{region "Read"}
5:
{region "Start Qiescent Mode"}
	fb103StartQuiescentMode(bStart := TRUE,
							eAddressType := Tc3_DALI.E_DALIAddressType.Broadcast,
							eCommandPriority := Tc3_DALI.E_DALICommandPriority.Middle);
	IF (NOT fb103StartQuiescentMode.bBusy) THEN
		fb103StartQuiescentMode(bStart := FALSE);
		nStep := 10;
	END_IF
{endregion}
10:
{region "Query Instance Error"}
	fb103QueryInstanceError(bStart := TRUE,
							nAddress := nAddress,
							eAddressType := Tc3_DALI.E_DALIAddressType.Short,
							nInstanceAddress := nInstanceAddress,
							eInstanceAddressType := Tc3_DALI.E_DALIInstanceAddressType.InstanceNumber,
							eCommandPriority := Tc3_DALI.E_DALICommandPriority.Middle,
							nInstanceError => nInstanceError);
	IF (NOT fb103QueryInstanceError.bBusy) THEN
		fb103QueryInstanceError(bStart := FALSE);
		nStep := 20;
	END_IF
{endregion}
20:
{region "Query Instance Status"}
	fb103QueryInstanceStatus(	bStart := TRUE,
								nAddress := nAddress,
								eAddressType := Tc3_DALI.E_DALIAddressType.Short,
								nInstanceAddress := nInstanceAddress,
								eInstanceAddressType := Tc3_DALI.E_DALIInstanceAddressType.InstanceNumber,
								eCommandPriority := Tc3_DALI.E_DALICommandPriority.Middle);
	IF (NOT fb103QueryInstanceStatus.bBusy) THEN
		fb103QueryInstanceStatus(bStart := FALSE);
		IF (fb103QueryInstanceStatus.nInstanceStatus.1) THEN
			bEnable := TRUE;
		END_IF
			nStep := 30;
	END_IF
30:
{region "Query Resolution"}
	fb103QueryResolution(	bStart := TRUE,
							nAddress := nAddress,
							eAddressType := Tc3_DALI.E_DALIAddressType.Short,
							nInstanceAddress := nInstanceAddress,
							eInstanceAddressType := Tc3_DALI.E_DALIInstanceAddressType.InstanceNumber,
							eCommandPriority := Tc3_DALI.E_DALICommandPriority.Middle,
							nResolution => nResolution);
	IF (NOT fb103QueryResolution.bBusy) THEN
		fb103QueryResolution(bStart := FALSE);
		nStep := 40;
	END_IF
{endregion}
40:
{region "Query Input Value"}
	fb103QueryInputValue(	bStart := TRUE,
							nAddress := nAddress,
							eAddressType:= Tc3_DALI.E_DALIAddressType.Short,
							nInstanceAddress := nInstanceAddress,
							eInstanceAddressType := Tc3_DALI.E_DALIInstanceAddressType.InstanceNumber,
							eCommandPriority := Tc3_DALI.E_DALICommandPriority.Middle,
							nResolution := nResolution,
							nInputValue => nInputValue);
	IF (NOT fb103QueryInputValue.bBusy) THEN
		fb103QueryInputValue(bStart := FALSE);
		nStep := 50;
	END_IF
{endregion}
50:
{region "Query Event Scheme"}
	fb103QueryEventScheme(	bStart := TRUE,
							nAddress := nAddress,
							eAddressType := Tc3_DALI.E_DALIAddressType.Short,
							nInstanceAddress := nInstanceAddress,
							eInstanceAddressType := Tc3_DALI.E_DALIInstanceAddressType.InstanceNumber,
							eCommandPriority := Tc3_DALI.E_DALICommandPriority.Middle,
							eEventScheme => eEventScheme);
	IF (NOT fb103QueryEventScheme.bBusy) THEN
		fb103QueryEventScheme(bStart := FALSE);
		nStep := 60;
	END_IF
{endregion}
60:
{region "Query Event Filter"}
	fb103QueryEventFilter(	bStart := TRUE,
							nAddress := nAddress,
							eAddressType := Tc3_DALI.E_DALIAddressType.Short,
							nInstanceAddress := nInstanceAddress,
							eInstanceAddressType := Tc3_DALI.E_DALIInstanceAddressType.InstanceNumber,
							eCommandPriority := Tc3_DALI.E_DALICommandPriority.Middle,
							nEventFilter => nEventFilter);
	IF (NOT fb103QueryEventFilter.bBusy) THEN
		fb103QueryEventFilter(bStart := FALSE);
		bPositionEventEnabled := nEventFilter.0;
		nStep := 70;
	END_IF
{endregion}
70:
{region "Query Report Timer"}
	fb302QueryReportTimer(	bStart := TRUE,
							nAddress := nAddress,
							eAddressType := Tc3_DALI.E_DALIAddressType.Short,
							nInstanceAddress := nInstanceAddress,
							eInstanceAddressType := Tc3_DALI.E_DALIInstanceAddressType.InstanceNumber,
							eCommandPriority := Tc3_DALI.E_DALICommandPriority.Middle,
							nReport => nReport);
	IF (NOT fb302QueryReportTimer.bBusy) THEN
		fb302QueryReportTimer(bStart := FALSE);
		nStep := 80;
	END_IF
{endregion}
80:
{region "Query Deadtime Timer"}
	fb302QueryDeadtimeTimer(bStart := TRUE,
							nAddress := nAddress,
							eAddressType := Tc3_DALI.E_DALIAddressType.Short,
							nInstanceAddress := nInstanceAddress,
							eInstanceAddressType := Tc3_DALI.E_DALIInstanceAddressType.InstanceNumber,
							eCommandPriority := Tc3_DALI.E_DALICommandPriority.Middle);
	nDeadtime := (fb302QueryDeadtimeTimer.nDeadtime * 50);
	IF (NOT fb302QueryDeadtimeTimer.bBusy) THEN
		fb302QueryDeadtimeTimer(bStart := FALSE);
		nStep := 90;
	END_IF
{endregion}
90:
	{region "Query Deadtime Timer"}
	fb302QuerySwitch(	bStart := TRUE,
						nAddress := nAddress,
						eAddressType := Tc3_DALI.E_DALIAddressType.Short,
						nInstanceAddress := nInstanceAddress,
						eInstanceAddressType := Tc3_DALI.E_DALIInstanceAddressType.InstanceNumber,
						eCommandPriority := Tc3_DALI.E_DALICommandPriority.Middle,
						bSwitch => bSwitch);
	IF (NOT fb302QueryDeadtimeTimer.bBusy) THEN
		fb302QueryDeadtimeTimer(bStart := FALSE);
		nStep := 100;
	END_IF
{endregion}
100:
{region "Query Event Priority"}
	fb103QueryEventPriority(bStart := TRUE,
							nAddress := nAddress,
							eAddressType := Tc3_DALI.E_DALIAddressType.Short,
							nInstanceAddress := nInstanceAddress,
							eInstanceAddressType := Tc3_DALI.E_DALIInstanceAddressType.InstanceNumber,
							eCommandPriority := Tc3_DALI.E_DALICommandPriority.Middle,
							eEventPriority => eEventPriority);
	IF (NOT fb103QueryEventPriority.bBusy) THEN
		fb103QueryEventPriority(bStart := FALSE);
		nStep := 110;
	END_IF 
{endregion}
110:
{region "Stop Qiescent Mode"}
	fb103StopQuiescentMode(	bStart := TRUE,
							eAddressType := Tc3_DALI.E_DALIAddressType.Broadcast,
							eCommandPriority := Tc3_DALI.E_DALICommandPriority.Middle);
	IF (NOT fb103StopQuiescentMode.bBusy) THEN
		fb103StopQuiescentMode(bStart := FALSE);
		nStep := 0;
	END_IF
{endregion}
{region "Write"}
1000:
{region "Enable or Disable Instance"}
	IF (bEnable) THEN
		fb103EnableInstance(bStart := TRUE,
							nAddress := nAddress,
							eAddressType := Tc3_DALI.E_DALIAddressType.Short,
							nInstanceAddress := nInstanceAddress,
							eInstanceAddressType := Tc3_DALI.E_DALIInstanceAddressType.InstanceNumber,
							eCommandPriority := Tc3_DALI.E_DALICommandPriority.Middle);
		IF (NOT fb103EnableInstance.bBusy) THEN
			fb103EnableInstance(bStart := FALSE);
			nStep := 1010;
		END_IF
	ELSE
		fb103DisableInstance(	bStart := TRUE,
								nAddress := nAddress,
								eAddressType := Tc3_DALI.E_DALIAddressType.Short,
								nInstanceAddress := nInstanceAddress,
								eInstanceAddressType := Tc3_DALI.E_DALIInstanceAddressType.InstanceNumber,
								eCommandPriority := Tc3_DALI.E_DALICommandPriority.Middle);
		IF (NOT fb103DisableInstance.bBusy) THEN
			fb103DisableInstance(bStart := FALSE);
			nStep := 0;
		END_IF
	END_IF
{endregion}
1010:
{region "Set Event Scheme"}
	fb103SetEventScheme(bStart := TRUE,
						nAddress := nAddress,
						eAddressType := Tc3_DALI.E_DALIAddressType.Short,
						nInstanceAddress := nInstanceAddress,
						eInstanceAddressType := Tc3_DALI.E_DALIInstanceAddressType.InstanceNumber,
						eCommandPriority := Tc3_DALI.E_DALICommandPriority.Middle,
						eEventScheme := eEventScheme);
	IF (NOT fb103SetEventScheme.bBusy) THEN
		fb103SetEventScheme(bStart := FALSE);
		nStep := 1020;
	END_IF
{endregion}
1020:
{region "Set Event Filter"}
	nEventFilter.0 := bPositionEventEnabled;
	fb103SetEventFilter(bStart := TRUE,
						nAddress := nAddress,
						eAddressType := Tc3_DALI.E_DALIAddressType.Short,
						nInstanceAddress := nInstanceAddress,
						eInstanceAddressType := Tc3_DALI.E_DALIInstanceAddressType.InstanceNumber,
						eCommandPriority := Tc3_DALI.E_DALICommandPriority.Middle,
						nEventFilter := nEventFilter);
	IF (NOT fb103SetEventFilter.bBusy) THEN
		fb103SetEventFilter(bStart := FALSE);
		nStep := 1030;
	END_IF
{endregion}
1030:
{region "Set Report Timer"}
	IF (bNoReportTimer) THEN
		nStep := 1040;
	ELSE
		fb302SetReportTimer(bStart := TRUE,
							nAddress := nAddress,
							eAddressType := Tc3_DALI.E_DALIAddressType.Short,
							nInstanceAddress := nInstanceAddress,
							eInstanceAddressType := Tc3_DALI.E_DALIInstanceAddressType.InstanceNumber,
							eCommandPriority := Tc3_DALI.E_DALICommandPriority.Middle,
							nReport := nReport);
		IF (NOT fb302SetReportTimer.bBusy) THEN
			fb302SetReportTimer(bStart := FALSE);
			nStep := 1040;
		END_IF
	END_IF
{endregion}
1040:
{region "Set Deadtime Timer"}
	IF (bNoDeadtimeTimer) THEN
		nStep := 1050;
	ELSE
		fb302SetDeadtimeTimer(	bStart := TRUE,
								nAddress := nAddress,
								eAddressType := Tc3_DALI.E_DALIAddressType.Short,
								nInstanceAddress := nInstanceAddress,
								eInstanceAddressType := Tc3_DALI.E_DALIInstanceAddressType.InstanceNumber,
								eCommandPriority := Tc3_DALI.E_DALICommandPriority.Middle,
								nDeadtime := TO_BYTE(nDeadtime / 50));
		IF (NOT fb302SetDeadtimeTimer.bBusy) THEN
			fb302SetDeadtimeTimer(bStart := FALSE);
			nStep := 1050;
		END_IF
	END_IF
{endregion}
1050:
{region "Set Event Priority"}
	fb103SetEventPriority(	bStart := TRUE,
							nAddress := nAddress,
							eAddressType := Tc3_DALI.E_DALIAddressType.Short,
							nInstanceAddress := nInstanceAddress,
							eInstanceAddressType := Tc3_DALI.E_DALIInstanceAddressType.InstanceNumber,
							eCommandPriority := Tc3_DALI.E_DALICommandPriority.Middle,
							eEventPriority := eEventPriority);
	IF (NOT fb103SetEventPriority.bBusy) THEN
		fb103SetEventPriority(bStart := FALSE);
		nStep := 0;
	END_IF
{endregion}
END_CASE
{endregion}

END_FUNCTION_BLOCK

// ---- POUs/DALI/DALI_Setup/FBs/FB_Part303OccupancySensor.TcPOU
FUNCTION_BLOCK FB_Part303OccupancySensor
VAR_INPUT
	ipDALICommunication			:	I_DALICommunication;
END_VAR
VAR_OUTPUT
	bBusy						:	BOOL;
END_VAR
VAR
{region "Visu"}
	sInputValue					:	STRING (50);
	nInstanceError				:	BYTE;
	nResolution					:	BYTE;
	eEventScheme				:	E_DALIEventScheme;
	nEventFilter				:	DWORD;
	nHold						:	UINT(1..2538);
	nHoldIntern					:	BYTE;
	nReport						:	BYTE(0..255);
	nDeadtime					:	UINT(0..12750);
	nDeadtimeIntern				:	BYTE;
	sCatching					:	STRING (20);
	bEnable						:	BOOL;
	bCancelHoldTimer			:	BOOL;
	bCatchmovement				:	BOOL;
	bRead						:	BOOL;
	bWrite						:	BOOL;
	bOccupied					:	BOOL;
	bVacant						:	BOOL;
	bRepeat						:	BOOL;
	bMovement					:	BOOL;
	bNoMovement					:	BOOL;
	bNoHoldTimer				:	BOOL;
	bNoReportTimer				:	BOOL;
	bNoDeadtimeTimer			:	BOOL;
	eEventPriority				:	E_DALIEventPriority := E_DALIEventPriority.MiddleLow;
{endregion}
	nStep						:	INT;
	nAddress					:	BYTE;
	nInstanceAddress			:	BYTE;
	bHideWaitSymbol				:	BOOL := TRUE;

	fb103StartQuiescentMode		:	FB_DALI103StartQuiescentMode(0);
	fb103StopQuiescentMode		:	FB_DALI103StopQuiescentMode(0);
	fb103QueryInstanceError		:	FB_DALI103QueryInstanceError(0);
	fb103QueryInstanceStatus	:	FB_DALI103QueryInstanceStatus(0);
	fb103QueryResolution		:	FB_DALI103QueryResolution(0);
	fb103QueryInputValue 		:	FB_DALI103QueryInputValue(0);
	fb103QueryEventScheme 		:	FB_DALI103QueryEventScheme(0);
	fb103QueryEventFilter 		:	FB_DALI103QueryEventFilter(0);
	fb103QueryEventPriority		:	FB_DALI103QueryEventPriority(0);
	fb303QueryCatching			:	FB_DALI303QueryCatching(0);
	fb303QueryHoldTimer			:	FB_DALI303QueryHoldTimer(0);
	fb303QueryReportTimer		:	FB_DALI303QueryReportTimer(0);
	fb303QueryDeadtimeTimer		:	FB_DALI303QueryDeadtimeTimer(0);
	fb103EnableInstance			:	FB_DALI103EnableInstance(0);
	fb103DisableInstance		:	FB_DALI103DisableInstance(0);
	fb103SetEventScheme			:	FB_DALI103SetEventScheme(0);
	fb103SetEventFilter			:	FB_DALI103SetEventFilter(0);
	fb103SetEventPriority		:	FB_DALI103SetEventPriority(0);
	fb303SetHoldTimer			:	FB_DALI303SetHoldTimer(0);
	fb303SetReportTimer			:	FB_DALI303SetReportTimer(0);
	fb303SetDeadtimeTimer		:	FB_DALI303SetDeadtimeTimer(0);
	fb303CancelHoldTimer		:	FB_DALI303CancelHoldTimer(0);
	fb303CatchMovement			:	FB_DALI303CatchMovement(0);
END_VAR

{region "Detect Commands"}
IF (bRead AND (nStep = 0)) THEN
	nStep := 5;
	bRead := FALSE;
	bHideWaitSymbol := FALSE;
END_IF

IF (bWrite AND (nStep = 0)) THEN
	nStep := 1000;
	bWrite := FALSE;
	bHideWaitSymbol := FALSE;
END_IF
{endregion}
{region "Manage Dialog Selection}
IF (nStep = 0) THEN
	bBusy := FALSE;
ELSE
	bBusy := TRUE;
END_IF
{endregion}
{region "Execute Commands"}
CASE nStep OF
0:
{region "Init"}
	bRead := FALSE;
	bWrite := FALSE;
	bHideWaitSymbol := TRUE;

	fb103StartQuiescentMode.ipDALICommunication := ipDALICommunication;
	fb103StopQuiescentMode.ipDALICommunication := ipDALICommunication;
	fb103QueryInstanceError.ipDALICommunication := ipDALICommunication;
	fb103QueryInstanceStatus.ipDALICommunication := ipDALICommunication;
	fb103QueryResolution.ipDALICommunication := ipDALICommunication;
	fb103QueryInputValue.ipDALICommunication := ipDALICommunication;
	fb103QueryEventScheme.ipDALICommunication := ipDALICommunication;
	fb103QueryEventFilter.ipDALICommunication := ipDALICommunication;
	fb103QueryEventPriority.ipDALICommunication := ipDALICommunication;
	fb303QueryCatching.ipDALICommunication := ipDALICommunication;
	fb303QueryHoldTimer.ipDALICommunication := ipDALICommunication;
	fb303QueryReportTimer.ipDALICommunication := ipDALICommunication;
	fb303QueryDeadtimeTimer.ipDALICommunication := ipDALICommunication;
	fb103EnableInstance.ipDALICommunication := ipDALICommunication;
	fb103DisableInstance.ipDALICommunication := ipDALICommunication;
	fb103SetEventScheme.ipDALICommunication := ipDALICommunication;
	fb103SetEventFilter.ipDALICommunication := ipDALICommunication;
	fb103SetEventPriority.ipDALICommunication := ipDALICommunication;
	fb303SetHoldTimer.ipDALICommunication := ipDALICommunication;
	fb303SetReportTimer.ipDALICommunication := ipDALICommunication;
	fb303SetDeadtimeTimer.ipDALICommunication := ipDALICommunication;
	fb303CancelHoldTimer.ipDALICommunication := ipDALICommunication;
	fb303CatchMovement.ipDALICommunication := ipDALICommunication;
{endregion}
{region "Read"}
5:
{region "Start Qiescent Mode"}
	fb103StartQuiescentMode(bStart := TRUE,
							eAddressType := Tc3_DALI.E_DALIAddressType.Broadcast,
							eCommandPriority := Tc3_DALI.E_DALICommandPriority.Middle);
	IF (NOT fb103StartQuiescentMode.bBusy) THEN
		fb103StartQuiescentMode(bStart:= FALSE);
		nStep := 10;
	END_IF
{endregion}
10:
{region "Query Instance Error"}
	fb103QueryInstanceError(bStart := TRUE,
							nAddress := nAddress,
							eAddressType := Tc3_DALI.E_DALIAddressType.Short,
							nInstanceAddress := nInstanceAddress,
							eInstanceAddressType := Tc3_DALI.E_DALIInstanceAddressType.InstanceNumber,
							eCommandPriority := Tc3_DALI.E_DALICommandPriority.Middle,
							nInstanceError => nInstanceError);
	IF (NOT fb103QueryInstanceError.bBusy) THEN
		fb103QueryInstanceError(bStart := FALSE);
		nStep := 20;
	END_IF
{endregion}
20:
{region "Query Instance Status"}
	fb103QueryInstanceStatus(	bStart := TRUE,
								nAddress := nAddress,
								eAddressType := Tc3_DALI.E_DALIAddressType.Short,
								nInstanceAddress := nInstanceAddress,
								eInstanceAddressType := Tc3_DALI.E_DALIInstanceAddressType.InstanceNumber,
								eCommandPriority := Tc3_DALI.E_DALICommandPriority.Middle);
	IF (NOT fb103QueryInstanceStatus.bBusy) THEN
		fb103QueryInstanceStatus(bStart := FALSE);
		IF (fb103QueryInstanceStatus.nInstanceStatus.1) THEN
			bEnable := TRUE;
		END_IF
		nStep := 30;
	END_IF
30:
{region "Query Resolution"}
	fb103QueryResolution(	bStart := TRUE,
							nAddress := nAddress,
							eAddressType := Tc3_DALI.E_DALIAddressType.Short,
							nInstanceAddress := nInstanceAddress,
							eInstanceAddressType := Tc3_DALI.E_DALIInstanceAddressType.InstanceNumber,
							eCommandPriority := Tc3_DALI.E_DALICommandPriority.Middle,
							nResolution => nResolution);
	IF (NOT fb103QueryResolution.bBusy) THEN
		fb103QueryResolution(bStart := FALSE);
		nStep := 40;
	END_IF
{endregion}
40:
{region "Query Input Value"}
	fb103QueryInputValue(	bStart := TRUE,
							nAddress := nAddress,
							eAddressType := Tc3_DALI.E_DALIAddressType.Short,
							nInstanceAddress := nInstanceAddress,
							eInstanceAddressType := Tc3_DALI.E_DALIInstanceAddressType.InstanceNumber,
							eCommandPriority := Tc3_DALI.E_DALICommandPriority.Middle,
							nResolution := nResolution);
	IF (NOT fb103QueryInputValue.bBusy) THEN
		fb103QueryInputValue(bStart:= FALSE);
		IF (fb103QueryInputValue.nInputValue = 0) THEN
			sInputValue := 'Vacant and no movement';
		ELSIF (fb103QueryInputValue.nInputValue = 1) THEN
			sInputValue := 'Vacant and movement';
		ELSIF (fb103QueryInputValue.nInputValue = 2) THEN
			sInputValue := 'Occupied and no movement';
		ELSIF (fb103QueryInputValue.nInputValue = 3) THEN
			sInputValue := 'Occupied and movement';
		END_IF
		nStep := 50;
	END_IF
{endregion}
50:
{region "Query Event Scheme"}
	fb103QueryEventScheme(	bStart := TRUE,
							nAddress := nAddress,
							eAddressType := Tc3_DALI.E_DALIAddressType.Short,
							nInstanceAddress := nInstanceAddress,
							eInstanceAddressType := Tc3_DALI.E_DALIInstanceAddressType.InstanceNumber,
							eCommandPriority := Tc3_DALI.E_DALICommandPriority.Middle,
							eEventScheme => eEventScheme);
	IF (NOT fb103QueryEventScheme.bBusy) THEN
		fb103QueryEventScheme(bStart := FALSE);
		nStep := 60;
	END_IF
{endregion}
60:
{region "Query Event Filter"}
	fb103QueryEventFilter(	bStart := TRUE,
							nAddress := nAddress,
							eAddressType := Tc3_DALI.E_DALIAddressType.Short,
							nInstanceAddress := nInstanceAddress,
							eInstanceAddressType := Tc3_DALI.E_DALIInstanceAddressType.InstanceNumber,
							eCommandPriority := Tc3_DALI.E_DALICommandPriority.Middle,
							nEventFilter => nEventFilter);
	IF (NOT fb103QueryEventFilter.bBusy) THEN
		fb103QueryEventFilter(bStart := FALSE);
		bOccupied := nEventFilter.0;
		bVacant := nEventFilter.1;
		bRepeat := nEventFilter.2;
		bMovement := nEventFilter.3;
		bNoMovement := nEventFilter.4;
		nStep := 70;
	END_IF
{endregion}
70: 
{region "Query Catching"}
	fb303QueryCatching(	bStart := TRUE,
						nAddress := nAddress,
						eAddressType := Tc3_DALI.E_DALIAddressType.Short,
						nInstanceAddress := nInstanceAddress,
						eInstanceAddressType := Tc3_DALI.E_DALIInstanceAddressType.InstanceNumber,
						eCommandPriority := Tc3_DALI.E_DALICommandPriority.Middle);
	IF (NOT fb303QueryCatching.bBusy) THEN
		fb303QueryCatching(bStart := FALSE);
		IF (fb303QueryCatching.bCatching) THEN
			sCatching := 'Active';
		ELSE
			sCatching := 'Inactive';
		END_IF
		nStep := 80;
	END_IF
80:
{region "Query Hold Timer"}
	fb303QueryHoldTimer(bStart := TRUE,
						nAddress := nAddress,
						eAddressType := Tc3_DALI.E_DALIAddressType.Short,
						nInstanceAddress := nInstanceAddress,
						eInstanceAddressType := Tc3_DALI.E_DALIInstanceAddressType.InstanceNumber,
						eCommandPriority := Tc3_DALI.E_DALICommandPriority.Middle,
						nHold => nHoldIntern);
	nHold := nHoldIntern * 10;
	IF (NOT fb303QueryHoldTimer.bBusy) THEN
		fb303QueryHoldTimer(bStart := FALSE);
		nStep := 90;
	END_IF
{endregion}
90:
{region "Query Report Timer"}
	fb303QueryReportTimer(	bStart := TRUE,
							nAddress := nAddress,
							eAddressType := Tc3_DALI.E_DALIAddressType.Short,
							nInstanceAddress := nInstanceAddress,
							eInstanceAddressType := Tc3_DALI.E_DALIInstanceAddressType.InstanceNumber,
							eCommandPriority := Tc3_DALI.E_DALICommandPriority.Middle,
							nReport => nReport);
	IF (NOT fb303QueryReportTimer.bBusy) THEN
		fb303QueryReportTimer(bStart := FALSE);
		nStep := 100;
	END_IF
{endregion}
100:
{region "Query Deadtime Timer"}
	fb303QueryDeadtimeTimer(bStart := TRUE,
							nAddress := nAddress,
							eAddressType := Tc3_DALI.E_DALIAddressType.Short,
							nInstanceAddress := nInstanceAddress,
							eInstanceAddressType := Tc3_DALI.E_DALIInstanceAddressType.InstanceNumber,
							eCommandPriority := Tc3_DALI.E_DALICommandPriority.Middle,
							nDeadtime => nDeadtimeIntern);
	nDeadtime := (nDeadtimeIntern * 50);
	IF (NOT fb303QueryDeadtimeTimer.bBusy) THEN
		fb303QueryDeadtimeTimer(bStart := FALSE);
		nStep := 110;
	END_IF
{endregion}
110:
{region "Query Event Priority"}
	fb103QueryEventPriority(bStart := TRUE,
							nAddress := nAddress,
							eAddressType := Tc3_DALI.E_DALIAddressType.Short,
							nInstanceAddress := nInstanceAddress,
							eInstanceAddressType := Tc3_DALI.E_DALIInstanceAddressType.InstanceNumber,
							eCommandPriority := Tc3_DALI.E_DALICommandPriority.Middle,
							eEventPriority => eEventPriority);
	IF (NOT fb103QueryEventPriority.bBusy) THEN
		fb103QueryEventPriority(bStart := FALSE);
		nStep := 120;
	END_IF 
{endregion}
120:
{region "Stop Qiescent Mode"}
	fb103StopQuiescentMode(	bStart:= TRUE,
							eAddressType:= Tc3_DALI.E_DALIAddressType.Broadcast,
							eCommandPriority:= Tc3_DALI.E_DALICommandPriority.Middle);
	IF (NOT fb103StopQuiescentMode.bBusy) THEN
		fb103StopQuiescentMode(bStart := FALSE);
		nStep := 0;
	END_IF
{endregion}

{region "Write"}
1000:
{region "Enable Instance"}
	IF (bEnable) THEN	
		fb103EnableInstance(bStart := TRUE,
							nAddress := nAddress,
							eAddressType := Tc3_DALI.E_DALIAddressType.Short,
							nInstanceAddress := nInstanceAddress,
							eInstanceAddressType := Tc3_DALI.E_DALIInstanceAddressType.InstanceNumber,
							eCommandPriority := Tc3_DALI.E_DALICommandPriority.Middle);
		IF (NOT fb103EnableInstance.bBusy) THEN
			fb103EnableInstance(bStart := FALSE);
			nStep := 1010;
		END_IF
	ELSE
		fb103DisableInstance(	bStart := TRUE,
								nAddress := nAddress,
								eAddressType := Tc3_DALI.E_DALIAddressType.Short,
								nInstanceAddress := nInstanceAddress,
								eInstanceAddressType := Tc3_DALI.E_DALIInstanceAddressType.InstanceNumber,
								eCommandPriority := Tc3_DALI.E_DALICommandPriority.Middle);
		IF (NOT fb103DisableInstance.bBusy) THEN
			fb103DisableInstance(bStart := FALSE);
			nStep := 0;
		END_IF
	END_IF
{endregion}
1010:
{region "Set Event Scheme"}
	fb103SetEventScheme(bStart := TRUE,
						nAddress := nAddress,
						eAddressType := Tc3_DALI.E_DALIAddressType.Short,
						nInstanceAddress := nInstanceAddress,
						eInstanceAddressType := Tc3_DALI.E_DALIInstanceAddressType.InstanceNumber,
						eCommandPriority := Tc3_DALI.E_DALICommandPriority.Middle,
						eEventScheme := eEventScheme);
	IF (NOT fb103SetEventScheme.bBusy) THEN
		fb103SetEventScheme(bStart := FALSE);
		nStep := 1020;
	END_IF
{endregion}
1020:
{region "Set Event Filter"}
	nEventFilter.0 := bOccupied;
	nEventFilter.1 := bVacant;
	nEventFilter.2 := bRepeat;
	nEventFilter.3 := bMovement;
	nEventFilter.4 := bNoMovement;
	fb103SetEventFilter(bStart := TRUE,
						nAddress := nAddress,
						eAddressType := Tc3_DALI.E_DALIAddressType.Short,
						nInstanceAddress := nInstanceAddress,
						eInstanceAddressType := Tc3_DALI.E_DALIInstanceAddressType.InstanceNumber,
						eCommandPriority := Tc3_DALI.E_DALICommandPriority.Middle,
						nEventFilter := nEventFilter);
	IF (NOT fb103SetEventFilter.bBusy) THEN
		fb103SetEventFilter(bStart := FALSE);
		nStep := 1030;
	END_IF
{endregion}
1030:
{region "Set Hold Timer"}
	IF (bNoHoldTimer) THEN
		nStep := 1040;
	ELSE
		fb303SetHoldTimer(	bStart := TRUE,
							nAddress := nAddress,
							eAddressType := Tc3_DALI.E_DALIAddressType.Short,
							nInstanceAddress := nInstanceAddress,
							eInstanceAddressType := Tc3_DALI.E_DALIInstanceAddressType.InstanceNumber,
							eCommandPriority := Tc3_DALI.E_DALICommandPriority.Middle,
							nHold := TO_BYTE(nHold / 10));
		IF (NOT fb303SetHoldTimer.bBusy) THEN
			fb303SetHoldTimer(bStart := FALSE);
			nStep := 1040;
		END_IF
	END_IF
{endregion}
1040:
{region "Set Report Timer"}
	IF (bNoReportTimer) THEN
		nStep := 1050;
	ELSE
		fb303SetReportTimer(bStart := TRUE,
							nAddress := nAddress,
							eAddressType := Tc3_DALI.E_DALIAddressType.Short,
							nInstanceAddress := nInstanceAddress,
							eInstanceAddressType := Tc3_DALI.E_DALIInstanceAddressType.InstanceNumber,
							eCommandPriority := Tc3_DALI.E_DALICommandPriority.Middle,
							nReport := nReport);
		IF (NOT fb303SetReportTimer.bBusy) THEN
			fb303SetReportTimer(bStart := FALSE);
			nStep := 1050;
		END_IF
	END_IF
{endregion}
1050:
{region "Set Deadtime Timer"}
	IF (bNoDeadtimeTimer) THEN
		nStep := 1060;
	ELSE
		fb303SetDeadtimeTimer(	bStart := TRUE,
								nAddress := nAddress,
								eAddressType := Tc3_DALI.E_DALIAddressType.Short,
								nInstanceAddress := nInstanceAddress,
								eInstanceAddressType := Tc3_DALI.E_DALIInstanceAddressType.InstanceNumber,
								eCommandPriority := Tc3_DALI.E_DALICommandPriority.Middle,
								nDeadtime := TO_BYTE(nDeadtime / 50));
		IF (NOT fb303SetDeadtimeTimer.bBusy) THEN
			fb303SetDeadtimeTimer(bStart := FALSE);
			nStep := 1060;
		END_IF
	END_IF
{endregion}
1060:
{region "Set Event Priority"}
	fb103SetEventPriority(	bStart := TRUE,
							nAddress := nAddress,
							eAddressType := Tc3_DALI.E_DALIAddressType.Short,
							nInstanceAddress := nInstanceAddress,
							eInstanceAddressType := Tc3_DALI.E_DALIInstanceAddressType.InstanceNumber,
							eCommandPriority := Tc3_DALI.E_DALICommandPriority.Middle,
							eEventPriority := eEventPriority);
	IF (NOT fb103SetEventPriority.bBusy) THEN
		fb103SetEventPriority(bStart := FALSE);
		nStep := 0;
	END_IF
{endregion}
END_CASE
{endregion}
{endregion}

{region "Cancel Hold Timer"}
IF (bCancelHoldTimer) THEN
	fb303CancelHoldTimer(bStart := TRUE);
END_IF
fb303CancelHoldTimer(	nAddress := nAddress,
						eAddressType := Tc3_DALI.E_DALIAddressType.Short,
						nInstanceAddress := nInstanceAddress,
						eInstanceAddressType := Tc3_DALI.E_DALIInstanceAddressType.InstanceNumber,
						eCommandPriority := Tc3_DALI.E_DALICommandPriority.Middle);
IF (NOT fb303CancelHoldTimer.bBusy) THEN
	bCancelHoldTimer := FALSE;
	fb303CancelHoldTimer(bStart := FALSE);
END_IF
{endregion}

{region "Catch Movement"}
IF (bCatchMovement) THEN
	fb303CatchMovement(bStart := TRUE);
END_IF
fb303CatchMovement(	nAddress := nAddress,
					eAddressType := Tc3_DALI.E_DALIAddressType.Short,
					nInstanceAddress := nInstanceAddress,
					eInstanceAddressType := Tc3_DALI.E_DALIInstanceAddressType.InstanceNumber,
					eCommandPriority := Tc3_DALI.E_DALICommandPriority.Middle);
IF (NOT fb303CatchMovement.bBusy) THEN
	bCatchMovement := FALSE;
	fb303CatchMovement(bStart := FALSE);
END_IF
{endregion}

END_FUNCTION_BLOCK

// ---- POUs/EnOcean/P_EnOcean.TcPOU
PROGRAM P_EnOcean
VAR
	fbKL6581			: FB_KL6581;
	stKL6581_in  AT %I* : KL6581_INPUT;
	stKL6581_out AT %Q*	: KL6581_OUTPUT;
	stKL6581			: STR_KL6581;
	bInitCom			: BOOL := TRUE;
	
	arrEnOcean_Search	: ARRAY [1..8] OF FB_EnOcean_Search;
	nSearchIdx			: BYTE;
	bSerach				: BOOL;
	arrDevices			: ARRAY [1..8] OF INT;
	arrID				: ARRAY [1..8, 0..255] OF DWORD;
	
		//Trykknapper Atrium
	fbAtriumNiveau_Tryk_PladeB				: FB_Rec_RPS_Switch;
	fbAtriumNiveau_Tryk_Sevice				: FB_Rec_RPS_Switch;			

	//Trykknapper på gange

	
	//Trykknapper i rum
	fbRum_2_449_Tryk					: FB_Rec_RPS_Switch;
	fbRum_3_461_Tryk					: FB_Rec_RPS_Switch;
	fbRum_3_463_Tryk					: FB_Rec_RPS_Switch;	
	fbRum_3_465_Tryk					: FB_Rec_RPS_Switch;

	
END_VAR

VAR CONSTANT
	byNode_1: BYTE := 1;
	byNode_2: BYTE := 2;
	byNode_3: BYTE := 3;
	byNode_4: BYTE := 4;
	byNode_5: BYTE := 5;
	byNode_6: BYTE := 6;
	byNode_7: BYTE := 7;
	byNode_8: BYTE := 8;
END_VAR


(* Kommunikation mit der KL6581. *)
(* Communication with the KL6581. *)
fbKL6581(
	bInit			:= bInitCom,
	nIdx			:= 2,
	stKL6581_in		:= stKL6581_In,
	stKL6581_out	:= stKL6581_Out,
	bReady			=> ,
	bBusy			=> ,
	bError			=> ,
	iErrorID		=> ,
	str_KL6581		=> stKL6581);

GVL_AHDataModbus.EnOceanError	:= TO_UINT(fbKL6581.iErrorID);
(* Warten bis der Kommunikationsbaustein initialisiert wurde.*)
(* Wait until the communication function block has been initialized. *)
IF (NOT fbKL6581.bReady) THEN
	RETURN;
END_IF

FOR nSearchIdx:= 1 TO 8 DO
	arrEnOcean_Search[nSearchIdx](
		bStart:= TRUE, 
		str_KL6581:= stKL6581 , 
		byNode:= nSearchIdx, 
		bReceive=> , 
		iDevices=>arrDevices[nSearchIdx] , 
		ar_ID=> );
		
		MEMCPY(ADR(arrID[nSearchIdx,0]), ADR(arrEnOcean_Search[nSearchIdx].ar_ID), SIZEOF(arrEnOcean_Search[nSearchIdx].ar_ID)); 
END_FOR

//A_Gang_3_364()

A_Rum_2_449();
A_Rum_3_461();
A_Rum_3_463();
A_Rum_3_465();

//AtriumNiveau
A_AtriumNiveau();

ACTION A_AtriumNiveau:
fbAtriumNiveau_Tryk_PladeB(
	str_KL6581:=stKL6581 , 
	byNode:=0, 
	dw_ID:= 16#0029B92D, 
	str_EnOceanSwitch=> GVL_EnOcean.strEnOceanSwitch_AtriumNiveau_PladeB,
	by_Node=> , 
	bReceive=> );
(*
fbAtriumNiveau_Tryk_Sevice(
	str_KL6581:=stKL6581 , 
	byNode:=0, 
	dw_ID:= 16#00FEE4FE87, 
	str_EnOceanSwitch=> GVL_EnOcean.strEnOceanSwitch_AtriumNiveau_Service, 
	by_Node=> , 
	bReceive=> );
*)
END_ACTION

ACTION A_Rum_2_449:
fbRum_2_449_Tryk(
	str_KL6581:=stKL6581 , 
	byNode:=0 , 
	dw_ID:= 16#0029ABAE, 
	str_EnOceanSwitch=> GVL_EnOcean.strEnOceanSwitch_Rum_2_449, 
	by_Node=> , 
	bReceive=> );
END_ACTION

ACTION A_Rum_3_461:
fbRum_3_461_Tryk(
	str_KL6581:=stKL6581 , 
	byNode:=0 , 
	dw_ID:= 16#0029AADB, 
	str_EnOceanSwitch=> GVL_EnOcean.strEnOceanSwitch_Rum_3_461, 
	by_Node=> , 
	bReceive=> );
END_ACTION

ACTION A_Rum_3_463:
fbRum_3_463_Tryk(
	str_KL6581:=stKL6581 , 
	byNode:=0 , 
	dw_ID:= 16#0029AACB, 
	str_EnOceanSwitch=> GVL_EnOcean.strEnOceanSwitch_Rum_3_463, 
	by_Node=> , 
	bReceive=> );
END_ACTION

ACTION A_Rum_3_465:
fbRum_3_465_Tryk(
	str_KL6581:=stKL6581 , 
	byNode:=0 , 
	dw_ID:= 16#0029AACE, 
	str_EnOceanSwitch=> GVL_EnOcean.strEnOceanSwitch_Rum_3_465, 
	by_Node=> , 
	bReceive=> );
END_ACTION

END_PROGRAM

// ---- POUs/MAIN.TcPOU
PROGRAM MAIN
VAR
	nAlive: INT;
	breset: BOOL;
	nDemoVariable : INT;
	nCX8200_State	AT %I*	: UINT;
END_VAR

VAR PERSISTENT
	nDemoVar_Persist: INT;
END_VAR

nAlive:= nAlive + 1;
GVL_AHDataModbus.nCX8200_State_MB := nCX8200_State;

P_SystemDK.M_nCyclic(bReset := breset );
P_DALI_DIAG();
DALI_Commissioning();
P_DALI_Energy_Line();
P_AHModbusComm();
P_DALI_Energy_Line();

//Gange
P_Gang_3_458();
P_Gang_3_409();
P_Gang_3_462A();

//Rum
P_Rum_2_449();
P_Rum_3_461();
P_Rum_3_463();
P_Rum_3_465();


//P_DALI_Energy_Firmware_Test();

END_PROGRAM

// ---- POUs/Alle_Rum/Gange/Gang_3_462A/Visualization_4_330.TcVIS
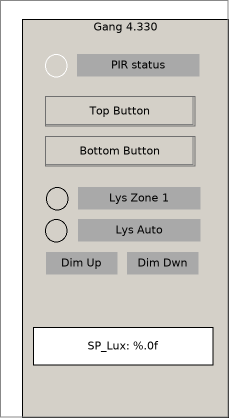
VISUALIZATION Visualization_4_330  // 229x418
    RoundedRectangle (22,19 207x399), "Gang 4.330"
    Rectangle (33,327 180x38), "SP_Lux: %.0f", text variable: P_Gang_3_462A.arrfbLysGruppe[1].fbLightCtrl.fLuxZone1
    Button (45,96 150x30), "Top Button"
        tap P_Gang_3_462A.bTopButtonZone1_Visu
    Button (45,136 150x30), "Bottom Button"
        tap P_Gang_3_462A.bBottomButtonZone1_Visu
    Ellipse (46,187 22x23), colour toggle: P_Gang_3_462A.fbLys.fbLightCtrl.bOnZone1
    Rectangle (78,187 122x22), "Lys Zone 1"
    Rectangle (46,252 71x22), "Dim Up", colour toggle: P_Gang_3_462A.arrfbLysGruppe[1].fbLightCtrl.bDimUp
    Rectangle (127,252 71x22), "Dim Dwn", colour toggle: P_Gang_3_462A.arrfbLysGruppe[1].fbLightCtrl.bDimDwn
    Ellipse (45,219 22x23), colour toggle: P_Gang_3_462A.arrfbLysGruppe[1].fbLightCtrl.bAutoZone1
    Rectangle (78,219 122x22), "Lys Auto"
    Ellipse (45,54 22x23), colour toggle: P_Gang_3_462A.arrfbLysGruppe[1].fbLightCtrl.bPIR
    Rectangle (77,54 122x22), "PIR status"
END_VISUALIZATION

// ---- POUs/Alle_Rum/Rum_Med_DALI_Pir/Rum_2_449/Visualization_5_356_1_2_1_1_1_1_1_1_1_1.TcVIS
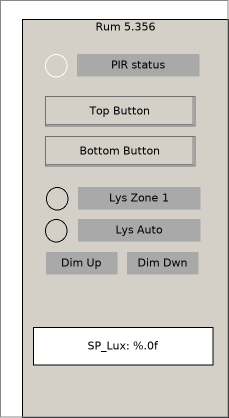
VISUALIZATION Visualization_5_356_1_2_1_1_1_1_1_1_1_1  // 229x418
    RoundedRectangle (22,19 207x399), "Rum 5.356"
    Rectangle (33,327 180x38), "SP_Lux: %.0f", text variable: P_Rum_5_356.arrfbLysGruppe[1].fbLightCtrl.fLuxZone1
    Button (45,96 150x30), "Top Button"
        tap P_Rum_5_356.bTopButtonZone1_Visu
    Button (45,136 150x30), "Bottom Button"
        tap P_Rum_5_356.bBottomButtonZone1_Visu
    Ellipse (46,187 22x23), colour toggle: P_Rum_5_356.arrfbLysGruppe[1].fbLightCtrl.bOnZone1
    Rectangle (78,187 122x22), "Lys Zone 1"
    Rectangle (46,252 71x22), "Dim Up", colour toggle: P_Rum_5_356.arrfbLysGruppe[1].fbLightCtrl.bDimUp
    Rectangle (127,252 71x22), "Dim Dwn", colour toggle: P_Rum_5_356.arrfbLysGruppe[1].fbLightCtrl.bDimDwn
    Ellipse (45,219 22x23), colour toggle: P_Rum_5_356.arrfbLysGruppe[1].fbLightCtrl.bAutoZone1
    Rectangle (78,219 122x22), "Lys Auto"
    Ellipse (45,54 22x23), colour toggle: P_Gang_5_356.arrfbLysGruppe[1].fbLightCtrl.bPIR
    Rectangle (77,54 122x22), "PIR status"
END_VISUALIZATION

// ---- POUs/Alle_Rum/Rum_Med_DALI_Pir/Rum_3_465/Visualization_5_e234.TcVIS
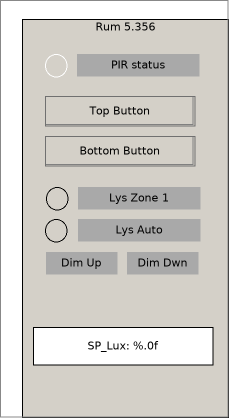
VISUALIZATION Visualization_5_e234  // 229x418
    RoundedRectangle (22,19 207x399), "Rum 5.356"
    Rectangle (33,327 180x38), "SP_Lux: %.0f", text variable: P_Rum_5_356.arrfbLysGruppe[1].fbLightCtrl.fLuxZone1
    Button (45,96 150x30), "Top Button"
        tap P_Rum_5_356.bTopButtonZone1_Visu
    Button (45,136 150x30), "Bottom Button"
        tap P_Rum_5_356.bBottomButtonZone1_Visu
    Ellipse (46,187 22x23), colour toggle: P_Rum_5_356.arrfbLysGruppe[1].fbLightCtrl.bOnZone1
    Rectangle (78,187 122x22), "Lys Zone 1"
    Rectangle (46,252 71x22), "Dim Up", colour toggle: P_Rum_5_356.arrfbLysGruppe[1].fbLightCtrl.bDimUp
    Rectangle (127,252 71x22), "Dim Dwn", colour toggle: P_Rum_5_356.arrfbLysGruppe[1].fbLightCtrl.bDimDwn
    Ellipse (45,219 22x23), colour toggle: P_Rum_5_356.arrfbLysGruppe[1].fbLightCtrl.bAutoZone1
    Rectangle (78,219 122x22), "Lys Auto"
    Ellipse (45,54 22x23), colour toggle: P_Gang_5_356.arrfbLysGruppe[1].fbLightCtrl.bPIR
    Rectangle (77,54 122x22), "PIR status"
END_VISUALIZATION

// ---- POUs/Alle_Rum/Rum_Med_DALI_Pir/Rum_3_463/Visualization_5_356.TcVIS
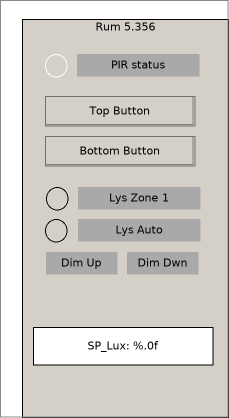
VISUALIZATION Visualization_5_356  // 229x418
    RoundedRectangle (22,19 207x399), "Rum 5.356"
    Rectangle (33,327 180x38), "SP_Lux: %.0f", text variable: P_Rum_5_356.arrfbLysGruppe[1].fbLightCtrl.fLuxZone1
    Button (45,96 150x30), "Top Button"
        tap P_Rum_5_356.bTopButtonZone1_Visu
    Button (45,136 150x30), "Bottom Button"
        tap P_Rum_5_356.bBottomButtonZone1_Visu
    Ellipse (46,187 22x23), colour toggle: P_Rum_5_356.arrfbLysGruppe[1].fbLightCtrl.bOnZone1
    Rectangle (78,187 122x22), "Lys Zone 1"
    Rectangle (46,252 71x22), "Dim Up", colour toggle: P_Rum_5_356.arrfbLysGruppe[1].fbLightCtrl.bDimUp
    Rectangle (127,252 71x22), "Dim Dwn", colour toggle: P_Rum_5_356.arrfbLysGruppe[1].fbLightCtrl.bDimDwn
    Ellipse (45,219 22x23), colour toggle: P_Rum_5_356.arrfbLysGruppe[1].fbLightCtrl.bAutoZone1
    Rectangle (78,219 122x22), "Lys Auto"
    Ellipse (45,54 22x23), colour toggle: P_Gang_5_356.arrfbLysGruppe[1].fbLightCtrl.bPIR
    Rectangle (77,54 122x22), "PIR status"
END_VISUALIZATION

// ---- POUs/Alle_Rum/Rum_Med_DALI_Pir/Rum_3_461/Visualization_5_352_1_1_1_1.TcVIS
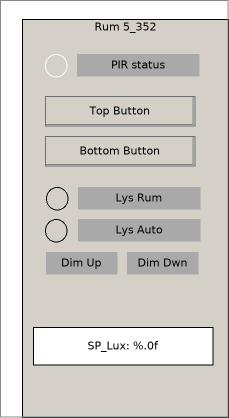
VISUALIZATION Visualization_5_352_1_1_1_1  // 229x418
    RoundedRectangle (22,19 207x399), "Rum 5_352"
    Rectangle (33,327 180x38), "SP_Lux: %.0f", text variable: P_Rum_4_324.fbLys.fbLightCtrl.fLuxZone1
    Button (45,96 150x30), "Top Button"
        tap P_Rum_5_352.bTopButtonZone1_Visu
    Button (45,136 150x30), "Bottom Button"
        tap P_Rum_5_352.bBottomButtonZone1_Visu
    Ellipse (46,187 22x23), colour toggle: P_Rum_5_352.fbLys.fbLightCtrl.bOnZone1
    Rectangle (78,187 122x22), "Lys Rum"
    Rectangle (46,252 71x22), "Dim Up", colour toggle: P_Rum_5_352.fbLys.fbLightCtrl.bDimUp
    Rectangle (127,252 71x22), "Dim Dwn", colour toggle: P_Rum_5_352.fbLys.fbLightCtrl.bDimDwn
    Ellipse (45,219 22x23), colour toggle: P_Rum_5_352.fbLys.fbLightCtrl.bAutoZone1
    Rectangle (78,219 122x22), "Lys Auto"
    Ellipse (45,54 22x23), colour toggle: P_Rum_5_352.fbLys.fbLightCtrl.bPIR
    Rectangle (77,54 122x22), "PIR status"
END_VISUALIZATION

// ---- POUs/DALI/DALI_Setup/VISUs/Visu_DALICommissioning.TcVIS
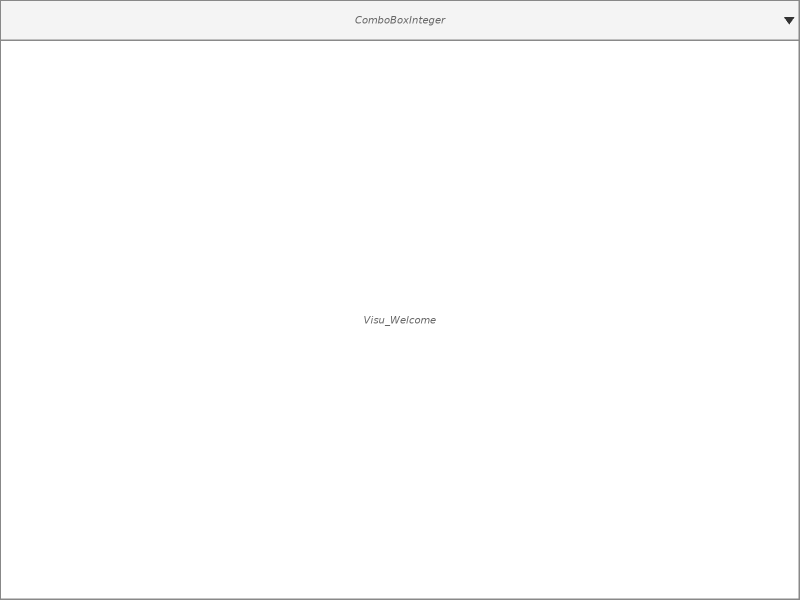
VISUALIZATION Visu_DALICommissioning  // 800x600
    ComboBoxInteger (0,0 800x40), variable: DALI_Commissioning.nSelectedDialog, input disabled if: DALI_Commissioning.bDisableComboBox, text list: 'TextList_Dialogs'
    Frame (0,40 800x560), frame switch variable: DALI_Commissioning.nSelectedDialog
        shows Visu_Welcome()
        shows Visu_Part102Commands()
        shows Visu_Part102Addressing()
        shows Visu_Part102Parameters()
        shows Visu_Part102Groups()
        shows Visu_Part102Scenes()
        shows Visu_Part102MemoryBank()
        shows Visu_Part102SetFading()
        shows Visu_Part202()
        shows Visu_Part205()
        shows Visu_Part207()
        shows Visu_Part208Switching()
        shows Visu_Part103Addressing()
        shows Visu_Part103Parameters()
        shows Visu_Part103Identify()
        shows Visu_Part301PushButton()
        shows Visu_Part302AbsoluteInputDevice()
        shows Visu_Part303OccupancySensor()
        shows Visu_Part304LightSensor()
        shows Visu_Part300GenericDevice()
        shows Visu_Part103MemoryBank()
        shows Visu_KL6821Configuration()
END_VISUALIZATION

// ---- POUs/DALI/DALI_Setup/VISUs/Visu_DALICommissioning/Visu_Part102Scenes.TcVIS
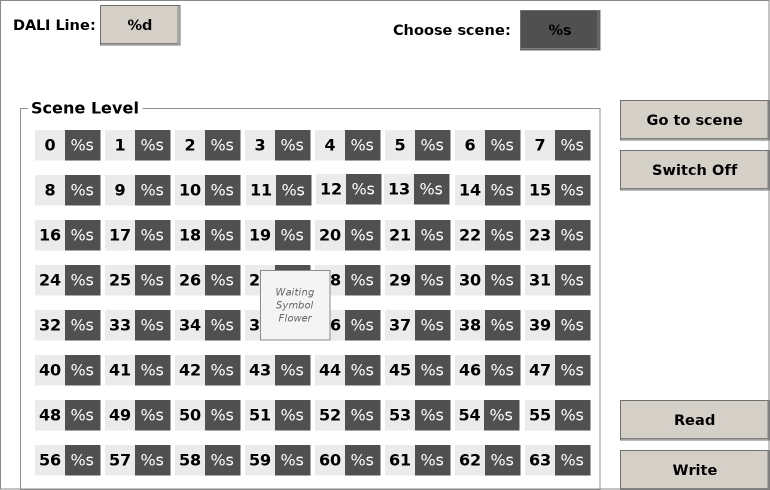
VISUALIZATION Visu_Part102Scenes  // 770x490
    GroupBox (20,100 580x390), "Scene Level"
        Group (85,30 65x30)
            Textfield (0,0 30x30), "1"
            Textfield (30,0 35x30), "%s", text variable: DALI_Commissioning.fbPart102Scenes.aScene[1], input disabled if: DALI_Commissioning.fbPart102Scenes.aNoShortAddress[1]
                p55702900: DALI_Commissioning.fbPart102Scenes.aFont[1]
                OnMouseClick: write the text variable via Default, min 0, max 255, title "Scene Value"
        Group (505,30 65x30)
            Textfield (0,0 30x30), "7"
            Textfield (30,0 35x30), "%s", text variable: DALI_Commissioning.fbPart102Scenes.aScene[7], input disabled if: DALI_Commissioning.fbPart102Scenes.aNoShortAddress[7]
                p55702900: DALI_Commissioning.fbPart102Scenes.aFont[7]
                OnMouseClick: write the text variable via Default, min 0, max 255, title "Scene Value"
        Group (435,30 65x30)
            Textfield (0,0 30x30), "6"
            Textfield (30,0 35x30), "%s", text variable: DALI_Commissioning.fbPart102Scenes.aScene[6], input disabled if: DALI_Commissioning.fbPart102Scenes.aNoShortAddress[6]
                p55702900: DALI_Commissioning.fbPart102Scenes.aFont[6]
                OnMouseClick: write the text variable via Default, min 0, max 255, title "Scene Value"
        Group (365,30 65x30)
            Textfield (0,0 30x30), "5"
            Textfield (30,0 35x30), "%s", text variable: DALI_Commissioning.fbPart102Scenes.aScene[5], input disabled if: DALI_Commissioning.fbPart102Scenes.aNoShortAddress[5]
                p55702900: DALI_Commissioning.fbPart102Scenes.aFont[5]
                OnMouseClick: write the text variable via Default, min 0, max 255, title "Scene Value"
        Group (295,30 65x30)
            Textfield (0,0 30x30), "4"
            Textfield (30,0 35x30), "%s", text variable: DALI_Commissioning.fbPart102Scenes.aScene[4], input disabled if: DALI_Commissioning.fbPart102Scenes.aNoShortAddress[4]
                p55702900: DALI_Commissioning.fbPart102Scenes.aFont[4]
                OnMouseClick: write the text variable via Default, min 0, max 255, title "Scene Value"
        Group (225,30 65x30)
            Textfield (0,0 30x30), "3"
            Textfield (30,0 35x30), "%s", text variable: DALI_Commissioning.fbPart102Scenes.aScene[3], input disabled if: DALI_Commissioning.fbPart102Scenes.aNoShortAddress[3]
                p55702900: DALI_Commissioning.fbPart102Scenes.aFont[3]
                OnMouseClick: write the text variable via Default, min 0, max 255, title "Scene Value"
        Group (155,30 65x30)
            Textfield (0,0 30x30), "2"
            Textfield (30,0 35x30), "%s", text variable: DALI_Commissioning.fbPart102Scenes.aScene[2], input disabled if: DALI_Commissioning.fbPart102Scenes.aNoShortAddress[2]
                p55702900: DALI_Commissioning.fbPart102Scenes.aFont[2]
                OnMouseClick: write the text variable via Default, min 0, max 255, title "Scene Value"
        Group (15,75 65x30)
            Textfield (0,0 30x30), "8"
            Textfield (30,0 35x30), "%s", text variable: DALI_Commissioning.fbPart102Scenes.aScene[8], input disabled if: DALI_Commissioning.fbPart102Scenes.aNoShortAddress[8]
                p55702900: DALI_Commissioning.fbPart102Scenes.aFont[8]
                OnMouseClick: write the text variable via Default, min 0, max 255, title "Scene Value"
        Group (15,120 65x30)
            Textfield (0,0 30x30), "16"
            Textfield (30,0 35x30), "%s", text variable: DALI_Commissioning.fbPart102Scenes.aScene[16], input disabled if: DALI_Commissioning.fbPart102Scenes.aNoShortAddress[16]
                p55702900: DALI_Commissioning.fbPart102Scenes.aFont[16]
                OnMouseClick: write the text variable via Default, min 0, max 255, title "Scene Value"
        Group (15,165 65x30)
            Textfield (0,0 30x30), "24"
            Textfield (30,0 35x30), "%s", text variable: DALI_Commissioning.fbPart102Scenes.aScene[24], input disabled if: DALI_Commissioning.fbPart102Scenes.aNoShortAddress[24]
                p55702900: DALI_Commissioning.fbPart102Scenes.aFont[24]
                OnMouseClick: write the text variable via Default, min 0, max 255, title "Scene Value"
        Group (15,210 65x30)
            Textfield (0,0 30x30), "32"
            Textfield (30,0 35x30), "%s", text variable: DALI_Commissioning.fbPart102Scenes.aScene[32], input disabled if: DALI_Commissioning.fbPart102Scenes.aNoShortAddress[32]
                p55702900: DALI_Commissioning.fbPart102Scenes.aFont[32]
                OnMouseClick: write the text variable via Default, min 0, max 255, title "Scene Value"
        Group (15,255 65x30)
            Textfield (0,0 30x30), "40"
            Textfield (30,0 35x30), "%s", text variable: DALI_Commissioning.fbPart102Scenes.aScene[40], input disabled if: DALI_Commissioning.fbPart102Scenes.aNoShortAddress[40]
                p55702900: DALI_Commissioning.fbPart102Scenes.aFont[40]
                OnMouseClick: write the text variable via Default, min 0, max 255, title "Scene Value"
        Group (15,300 65x30)
            Textfield (0,0 30x30), "48"
            Textfield (30,0 35x30), "%s", text variable: DALI_Commissioning.fbPart102Scenes.aScene[48], input disabled if: DALI_Commissioning.fbPart102Scenes.aNoShortAddress[48]
                p55702900: DALI_Commissioning.fbPart102Scenes.aFont[48]
                OnMouseClick: write the text variable via Default, min 0, max 255, title "Scene Value"
        Group (15,345 65x30)
            Textfield (0,0 30x30), "56"
            Textfield (30,0 35x30), "%s", text variable: DALI_Commissioning.fbPart102Scenes.aScene[56], input disabled if: DALI_Commissioning.fbPart102Scenes.aNoShortAddress[56]
                p55702900: DALI_Commissioning.fbPart102Scenes.aFont[56]
                OnMouseClick: write the text variable via Default, min 0, max 255, title "Scene Value"
        Group (85,75 65x30)
            Textfield (0,0 30x30), "9"
            Textfield (30,0 35x30), "%s", text variable: DALI_Commissioning.fbPart102Scenes.aScene[9], input disabled if: DALI_Commissioning.fbPart102Scenes.aNoShortAddress[9]
                p55702900: DALI_Commissioning.fbPart102Scenes.aFont[9]
                OnMouseClick: write the text variable via Default, min 0, max 255, title "Scene Value"
        Group (155,75 65x30)
            Textfield (0,0 30x30), "10"
            Textfield (30,0 35x30), "%s", text variable: DALI_Commissioning.fbPart102Scenes.aScene[10], input disabled if: DALI_Commissioning.fbPart102Scenes.aNoShortAddress[10]
                p55702900: DALI_Commissioning.fbPart102Scenes.aFont[10]
                OnMouseClick: write the text variable via Default, min 0, max 255, title "Scene Value"
        Group (226,75 65x30)
            Textfield (0,0 30x30), "11"
            Textfield (30,0 35x30), "%s", text variable: DALI_Commissioning.fbPart102Scenes.aScene[11], input disabled if: DALI_Commissioning.fbPart102Scenes.aNoShortAddress[11]
                p55702900: DALI_Commissioning.fbPart102Scenes.aFont[11]
                OnMouseClick: write the text variable via Default, min 0, max 255, title "Scene Value"
        Group (296,74 65x30)
            Textfield (0,0 30x30), "12"
            Textfield (30,0 35x30), "%s", text variable: DALI_Commissioning.fbPart102Scenes.aScene[12], input disabled if: DALI_Commissioning.fbPart102Scenes.aNoShortAddress[12]
                p55702900: DALI_Commissioning.fbPart102Scenes.aFont[12]
                OnMouseClick: write the text variable via Default, min 0, max 255, title "Scene Value"
        Group (364,74 65x30)
            Textfield (0,0 30x30), "13"
            Textfield (30,0 35x30), "%s", text variable: DALI_Commissioning.fbPart102Scenes.aScene[13], input disabled if: DALI_Commissioning.fbPart102Scenes.aNoShortAddress[13]
                p55702900: DALI_Commissioning.fbPart102Scenes.aFont[13]
                OnMouseClick: write the text variable via Default, min 0, max 255, title "Scene Value"
        Group (435,75 65x30)
            Textfield (0,0 30x30), "14"
            Textfield (30,0 35x30), "%s", text variable: DALI_Commissioning.fbPart102Scenes.aScene[14], input disabled if: DALI_Commissioning.fbPart102Scenes.aNoShortAddress[14]
                p55702900: DALI_Commissioning.fbPart102Scenes.aFont[14]
                OnMouseClick: write the text variable via Default, min 0, max 255, title "Scene Value"
        Group (505,75 65x30)
            Textfield (0,0 30x30), "15"
            Textfield (30,0 35x30), "%s", text variable: DALI_Commissioning.fbPart102Scenes.aScene[15], input disabled if: DALI_Commissioning.fbPart102Scenes.aNoShortAddress[15]
                p55702900: DALI_Commissioning.fbPart102Scenes.aFont[15]
                OnMouseClick: write the text variable via Default, min 0, max 255, title "Scene Value"
        Group (85,120 65x30)
            Textfield (0,0 30x30), "17"
            Textfield (30,0 35x30), "%s", text variable: DALI_Commissioning.fbPart102Scenes.aScene[17], input disabled if: DALI_Commissioning.fbPart102Scenes.aNoShortAddress[17]
                p55702900: DALI_Commissioning.fbPart102Scenes.aFont[17]
                OnMouseClick: write the text variable via Default, min 0, max 255, title "Scene Value"
        Group (155,120 65x30)
            Textfield (0,0 30x30), "18"
            Textfield (30,0 35x30), "%s", text variable: DALI_Commissioning.fbPart102Scenes.aScene[18], input disabled if: DALI_Commissioning.fbPart102Scenes.aNoShortAddress[18]
                p55702900: DALI_Commissioning.fbPart102Scenes.aFont[18]
                OnMouseClick: write the text variable via Default, min 0, max 255, title "Scene Value"
        Group (225,120 65x30)
            Textfield (0,0 30x30), "19"
            Textfield (30,0 35x30), "%s", text variable: DALI_Commissioning.fbPart102Scenes.aScene[19], input disabled if: DALI_Commissioning.fbPart102Scenes.aNoShortAddress[19]
                p55702900: DALI_Commissioning.fbPart102Scenes.aFont[19]
                OnMouseClick: write the text variable via Default, min 0, max 255, title "Scene Value"
        Group (295,120 65x30)
            Textfield (0,0 30x30), "20"
            Textfield (30,0 35x30), "%s", text variable: DALI_Commissioning.fbPart102Scenes.aScene[20], input disabled if: DALI_Commissioning.fbPart102Scenes.aNoShortAddress[20]
                p55702900: DALI_Commissioning.fbPart102Scenes.aFont[20]
                OnMouseClick: write the text variable via Default, min 0, max 255, title "Scene Value"
        Group (365,120 65x30)
            Textfield (0,0 30x30), "21"
            Textfield (30,0 35x30), "%s", text variable: DALI_Commissioning.fbPart102Scenes.aScene[21], input disabled if: DALI_Commissioning.fbPart102Scenes.aNoShortAddress[21]
                p55702900: DALI_Commissioning.fbPart102Scenes.aFont[21]
                OnMouseClick: write the text variable via Default, min 0, max 255, title "Scene Value"
        Group (435,120 65x30)
            Textfield (0,0 30x30), "22"
            Textfield (30,0 35x30), "%s", text variable: DALI_Commissioning.fbPart102Scenes.aScene[22], input disabled if: DALI_Commissioning.fbPart102Scenes.aNoShortAddress[22]
                p55702900: DALI_Commissioning.fbPart102Scenes.aFont[22]
                OnMouseClick: write the text variable via Default, min 0, max 255, title "Scene Value"
        Group (505,120 65x30)
            Textfield (0,0 30x30), "23"
            Textfield (30,0 35x30), "%s", text variable: DALI_Commissioning.fbPart102Scenes.aScene[23], input disabled if: DALI_Commissioning.fbPart102Scenes.aNoShortAddress[23]
                p55702900: DALI_Commissioning.fbPart102Scenes.aFont[23]
                OnMouseClick: write the text variable via Default, min 0, max 255, title "Scene Value"
        Group (85,165 65x30)
            Textfield (0,0 30x30), "25"
            Textfield (30,0 35x30), "%s", text variable: DALI_Commissioning.fbPart102Scenes.aScene[25], input disabled if: DALI_Commissioning.fbPart102Scenes.aNoShortAddress[25]
                p55702900: DALI_Commissioning.fbPart102Scenes.aFont[25]
                OnMouseClick: write the text variable via Default, min 0, max 255, title "Scene Value"
        Group (155,165 65x30)
            Textfield (0,0 30x30), "26"
            Textfield (30,0 35x30), "%s", text variable: DALI_Commissioning.fbPart102Scenes.aScene[26], input disabled if: DALI_Commissioning.fbPart102Scenes.aNoShortAddress[26]
                p55702900: DALI_Commissioning.fbPart102Scenes.aFont[26]
                OnMouseClick: write the text variable via Default, min 0, max 255, title "Scene Value"
        Group (225,165 65x30)
            Textfield (0,0 30x30), "27"
            Textfield (30,0 35x30), "%s", text variable: DALI_Commissioning.fbPart102Scenes.aScene[27], input disabled if: DALI_Commissioning.fbPart102Scenes.aNoShortAddress[27]
                p55702900: DALI_Commissioning.fbPart102Scenes.aFont[27]
                OnMouseClick: write the text variable via Default, min 0, max 255, title "Scene Value"
        Group (295,165 65x30)
            Textfield (0,0 30x30), "28"
            Textfield (30,0 35x30), "%s", text variable: DALI_Commissioning.fbPart102Scenes.aScene[28], input disabled if: DALI_Commissioning.fbPart102Scenes.aNoShortAddress[28]
                p55702900: DALI_Commissioning.fbPart102Scenes.aFont[28]
                OnMouseClick: write the text variable via Default, min 0, max 255, title "Scene Value"
        Group (365,165 65x30)
            Textfield (0,0 30x30), "29"
            Textfield (30,0 35x30), "%s", text variable: DALI_Commissioning.fbPart102Scenes.aScene[29], input disabled if: DALI_Commissioning.fbPart102Scenes.aNoShortAddress[29]
                p55702900: DALI_Commissioning.fbPart102Scenes.aFont[29]
                OnMouseClick: write the text variable via Default, min 0, max 255, title "Scene Value"
        Group (435,165 65x30)
            Textfield (0,0 30x30), "30"
            Textfield (30,0 35x30), "%s", text variable: DALI_Commissioning.fbPart102Scenes.aScene[30], input disabled if: DALI_Commissioning.fbPart102Scenes.aNoShortAddress[30]
                p55702900: DALI_Commissioning.fbPart102Scenes.aFont[30]
                OnMouseClick: write the text variable via Default, min 0, max 255, title "Scene Value"
        Group (505,165 65x30)
            Textfield (0,0 30x30), "31"
            Textfield (30,0 35x30), "%s", text variable: DALI_Commissioning.fbPart102Scenes.aScene[31], input disabled if: DALI_Commissioning.fbPart102Scenes.aNoShortAddress[31]
                p55702900: DALI_Commissioning.fbPart102Scenes.aFont[31]
                OnMouseClick: write the text variable via Default, min 0, max 255, title "Scene Value"
        Group (85,210 65x30)
            Textfield (0,0 30x30), "33"
            Textfield (30,0 35x30), "%s", text variable: DALI_Commissioning.fbPart102Scenes.aScene[33], input disabled if: DALI_Commissioning.fbPart102Scenes.aNoShortAddress[32]
                p55702900: DALI_Commissioning.fbPart102Scenes.aFont[33]
                OnMouseClick: write the text variable via Default, min 0, max 255, title "Scene Value"
        Group (155,210 65x30)
            Textfield (0,0 30x30), "34"
            Textfield (30,0 35x30), "%s", text variable: DALI_Commissioning.fbPart102Scenes.aScene[34], input disabled if: DALI_Commissioning.fbPart102Scenes.aNoShortAddress[34]
                p55702900: DALI_Commissioning.fbPart102Scenes.aFont[34]
                OnMouseClick: write the text variable via Default, min 0, max 255, title "Scene Value"
        Group (295,210 65x30)
            Textfield (0,0 30x30), "36"
            Textfield (30,0 35x30), "%s", text variable: DALI_Commissioning.fbPart102Scenes.aScene[36], input disabled if: DALI_Commissioning.fbPart102Scenes.aNoShortAddress[36]
                p55702900: DALI_Commissioning.fbPart102Scenes.aFont[36]
                OnMouseClick: write the text variable via Default, min 0, max 255
        Group (365,210 65x30)
            Textfield (0,0 30x30), "37"
            Textfield (30,0 35x30), "%s", text variable: DALI_Commissioning.fbPart102Scenes.aScene[37], input disabled if: DALI_Commissioning.fbPart102Scenes.aNoShortAddress[37]
                p55702900: DALI_Commissioning.fbPart102Scenes.aFont[37]
                OnMouseClick: write the text variable via Default, min 0, max 255, title "Scene Value"
        Group (435,210 65x30)
            Textfield (0,0 30x30), "38"
            Textfield (30,0 35x30), "%s", text variable: DALI_Commissioning.fbPart102Scenes.aScene[38], input disabled if: DALI_Commissioning.fbPart102Scenes.aNoShortAddress[38]
                p55702900: DALI_Commissioning.fbPart102Scenes.aFont[38]
                OnMouseClick: write the text variable via Default, min 0, max 255, title "Scene Value"
        Group (505,210 65x30)
            Textfield (0,0 30x30), "39"
            Textfield (30,0 35x30), "%s", text variable: DALI_Commissioning.fbPart102Scenes.aScene[39], input disabled if: DALI_Commissioning.fbPart102Scenes.aNoShortAddress[39]
                p55702900: DALI_Commissioning.fbPart102Scenes.aFont[39]
                OnMouseClick: write the text variable via Default, min 0, max 255, title "Scene Value"
        Group (85,255 65x30)
            Textfield (0,0 30x30), "41"
            Textfield (30,0 35x30), "%s", text variable: DALI_Commissioning.fbPart102Scenes.aScene[41], input disabled if: DALI_Commissioning.fbPart102Scenes.aNoShortAddress[41]
                p55702900: DALI_Commissioning.fbPart102Scenes.aFont[41]
                OnMouseClick: write the text variable via Default, min 0, max 255, title "Scene Value"
        Group (155,255 65x30)
            Textfield (0,0 30x30), "42"
            Textfield (30,0 35x30), "%s", text variable: DALI_Commissioning.fbPart102Scenes.aScene[42], input disabled if: DALI_Commissioning.fbPart102Scenes.aNoShortAddress[42]
                p55702900: DALI_Commissioning.fbPart102Scenes.aFont[42]
                OnMouseClick: write the text variable via Default, min 0, max 255, title "Scene Value"
        Group (225,210 65x30)
            Textfield (0,0 30x30), "35"
            Textfield (30,0 35x30), "%s", text variable: DALI_Commissioning.fbPart102Scenes.aScene[35], input disabled if: DALI_Commissioning.fbPart102Scenes.aNoShortAddress[35]
                p55702900: DALI_Commissioning.fbPart102Scenes.aFont[35]
                OnMouseClick: write the text variable via Default, min 0, max 255, title "Scene Value"
        Group (225,255 65x30)
            Textfield (0,0 30x30), "43"
            Textfield (30,0 35x30), "%s", text variable: DALI_Commissioning.fbPart102Scenes.aScene[43], input disabled if: DALI_Commissioning.fbPart102Scenes.aNoShortAddress[43]
                p55702900: DALI_Commissioning.fbPart102Scenes.aFont[43]
                OnMouseClick: write the text variable via Default, min 0, max 255, title "Scene Value"
        Group (295,255 65x30)
            Textfield (0,0 30x30), "44"
            Textfield (30,0 35x30), "%s", text variable: DALI_Commissioning.fbPart102Scenes.aScene[44], input disabled if: DALI_Commissioning.fbPart102Scenes.aNoShortAddress[44]
                p55702900: DALI_Commissioning.fbPart102Scenes.aFont[44]
                OnMouseClick: write the text variable via Default, min 0, max 255, title "Scene Value"
        Group (365,255 65x30)
            Textfield (0,0 30x30), "45"
            Textfield (30,0 35x30), "%s", text variable: DALI_Commissioning.fbPart102Scenes.aScene[45], input disabled if: DALI_Commissioning.fbPart102Scenes.aNoShortAddress[45]
                p55702900: DALI_Commissioning.fbPart102Scenes.aFont[45]
                OnMouseClick: write the text variable via Default, min 0, max 255, title "Scene Value"
        Group (435,255 65x30)
            Textfield (0,0 30x30), "46"
            Textfield (30,0 35x30), "%s", text variable: DALI_Commissioning.fbPart102Scenes.aScene[46], input disabled if: DALI_Commissioning.fbPart102Scenes.aNoShortAddress[46]
                p55702900: DALI_Commissioning.fbPart102Scenes.aFont[46]
                OnMouseClick: write the text variable via Default, min 0, max 255, title "Scene Value"
        Group (505,255 65x30)
            Textfield (0,0 30x30), "47"
            Textfield (30,0 35x30), "%s", text variable: DALI_Commissioning.fbPart102Scenes.aScene[47], input disabled if: DALI_Commissioning.fbPart102Scenes.aNoShortAddress[47]
                p55702900: DALI_Commissioning.fbPart102Scenes.aFont[47]
                OnMouseClick: write the text variable via Default, min 0, max 255, title "Scene Value"
        Group (85,300 65x30)
            Textfield (0,0 30x30), "49"
            Textfield (30,0 35x30), "%s", text variable: DALI_Commissioning.fbPart102Scenes.aScene[49], input disabled if: DALI_Commissioning.fbPart102Scenes.aNoShortAddress[49]
                p55702900: DALI_Commissioning.fbPart102Scenes.aFont[49]
                OnMouseClick: write the text variable via Default, min 0, max 255, title "Scene Value"
        Group (155,300 65x30)
            Textfield (0,0 30x30), "50"
            Textfield (30,0 35x30), "%s", text variable: DALI_Commissioning.fbPart102Scenes.aScene[50], input disabled if: DALI_Commissioning.fbPart102Scenes.aNoShortAddress[50]
                p55702900: DALI_Commissioning.fbPart102Scenes.aFont[50]
                OnMouseClick: write the text variable via Default, min 0, max 255, title "Scene Value"
        Group (225,300 65x30)
            Textfield (0,0 30x30), "51"
            Textfield (30,0 35x30), "%s", text variable: DALI_Commissioning.fbPart102Scenes.aScene[51], input disabled if: DALI_Commissioning.fbPart102Scenes.aNoShortAddress[51]
                p55702900: DALI_Commissioning.fbPart102Scenes.aFont[51]
                OnMouseClick: write the text variable via Default, min 0, max 255, title "Scene Value"
        Group (295,300 65x30)
            Textfield (0,0 30x30), "52"
            Textfield (30,0 35x30), "%s", text variable: DALI_Commissioning.fbPart102Scenes.aScene[52], input disabled if: DALI_Commissioning.fbPart102Scenes.aNoShortAddress[52]
                p55702900: DALI_Commissioning.fbPart102Scenes.aFont[52]
                OnMouseClick: write the text variable via Default, min 0, max 255, title "Scene Value"
        Group (365,300 65x30)
            Textfield (0,0 30x30), "53"
            Textfield (30,0 35x30), "%s", text variable: DALI_Commissioning.fbPart102Scenes.aScene[53], input disabled if: DALI_Commissioning.fbPart102Scenes.aNoShortAddress[53]
                p55702900: DALI_Commissioning.fbPart102Scenes.aFont[53]
                OnMouseClick: write the text variable via Default, min 0, max 255, title "Scene Value"
        Group (435,300 64x30)
            Textfield (0,0 29x30), "54"
            Textfield (29,0 35x30), "%s", text variable: DALI_Commissioning.fbPart102Scenes.aScene[54], input disabled if: DALI_Commissioning.fbPart102Scenes.aNoShortAddress[54]
                p55702900: DALI_Commissioning.fbPart102Scenes.aFont[54]
                OnMouseClick: write the text variable via Default, min 0, max 255, title "Scene Value"
        Group (505,300 65x30)
            Textfield (0,0 30x30), "55"
            Textfield (30,0 35x30), "%s", text variable: DALI_Commissioning.fbPart102Scenes.aScene[55], input disabled if: DALI_Commissioning.fbPart102Scenes.aNoShortAddress[55]
                p55702900: DALI_Commissioning.fbPart102Scenes.aFont[55]
                OnMouseClick: write the text variable via Default, min 0, max 255, title "Scene Value"
        Group (85,345 65x30)
            Textfield (0,0 30x30), "57"
            Textfield (30,0 35x30), "%s", text variable: DALI_Commissioning.fbPart102Scenes.aScene[57], input disabled if: DALI_Commissioning.fbPart102Scenes.aNoShortAddress[57]
                p55702900: DALI_Commissioning.fbPart102Scenes.aFont[57]
                OnMouseClick: write the text variable via Default, min 0, max 255, title "Scene Value"
        Group (155,345 65x30)
            Textfield (0,0 30x30), "58"
            Textfield (30,0 35x30), "%s", text variable: DALI_Commissioning.fbPart102Scenes.aScene[58], input disabled if: DALI_Commissioning.fbPart102Scenes.aNoShortAddress[58]
                p55702900: DALI_Commissioning.fbPart102Scenes.aFont[58]
                OnMouseClick: write the text variable via Default, min 0, max 255, title "Scene Value"
        Group (225,345 65x30)
            Textfield (0,0 30x30), "59"
            Textfield (30,0 35x30), "%s", text variable: DALI_Commissioning.fbPart102Scenes.aScene[59], input disabled if: DALI_Commissioning.fbPart102Scenes.aNoShortAddress[59]
                p55702900: DALI_Commissioning.fbPart102Scenes.aFont[59]
                OnMouseClick: write the text variable via Default, min 0, max 255, title "Scene Value"
        Group (295,345 65x30)
            Textfield (0,0 30x30), "60"
            Textfield (30,0 35x30), "%s", text variable: DALI_Commissioning.fbPart102Scenes.aScene[60], input disabled if: DALI_Commissioning.fbPart102Scenes.aNoShortAddress[60]
                p55702900: DALI_Commissioning.fbPart102Scenes.aFont[60]
                OnMouseClick: write the text variable via Default, min 0, max 255, title "Scene Value"
        Group (365,345 65x30)
            Textfield (0,0 30x30), "61"
            Textfield (30,0 35x30), "%s", text variable: DALI_Commissioning.fbPart102Scenes.aScene[61], input disabled if: DALI_Commissioning.fbPart102Scenes.aNoShortAddress[61]
                p55702900: DALI_Commissioning.fbPart102Scenes.aFont[61]
                OnMouseClick: write the text variable via Default, min 0, max 255, title "Scene Value"
        Group (435,345 65x30)
            Textfield (0,0 30x30), "62"
            Textfield (30,0 35x30), "%s", text variable: DALI_Commissioning.fbPart102Scenes.aScene[62], input disabled if: DALI_Commissioning.fbPart102Scenes.aNoShortAddress[62]
                p55702900: DALI_Commissioning.fbPart102Scenes.aFont[62]
                OnMouseClick: write the text variable via Default, min 0, max 255, title "Scene Value"
        Group (505,345 65x30)
            Textfield (0,0 30x30), "63"
            Textfield (30,0 35x30), "%s", text variable: DALI_Commissioning.fbPart102Scenes.aScene[63], input disabled if: DALI_Commissioning.fbPart102Scenes.aNoShortAddress[63]
                p55702900: DALI_Commissioning.fbPart102Scenes.aFont[63]
                OnMouseClick: write the text variable via Default, min 0, max 255, title "Scene Value"
        WaitingSymbolFlower (240,170 70x70), invisible if: DALI_Commissioning.fbPart102Scenes.bHideWaitSymbol
        Group (15,30 65x30)
            Textfield (0,0 30x30), "0"
            Textfield (30,0 35x30), "%s", text variable: DALI_Commissioning.fbPart102Scenes.aScene[0], input disabled if: DALI_Commissioning.fbPart102Scenes.aNoShortAddress[0]
                p55702900: DALI_Commissioning.fbPart102Scenes.aFont[0]
                OnMouseClick: write the text variable via Default, min 0, max 255, title "Scene Value"
    Button (620,400 150x40), "Read"
        OnMouseClick: execute { DALI_Commissioning.fbPart102Scenes.bRead := TRUE; }
    Button (620,450 150x40), "Write"
        OnMouseClick: execute { DALI_Commissioning.fbPart102Scenes.bWrite := TRUE; }
    Button (620,100 150x40), "Go to scene"
        OnMouseClick: execute { DALI_Commissioning.fbPart102Scenes.bGoToScene := TRUE; }
    Button (620,150 150x40), "Switch Off"
        OnMouseClick: execute { DALI_Commissioning.fbPart102Scenes.bSwitchOff := TRUE; }
    Textfield (390,10 120x40), "Choose scene:"
    Button (520,10 80x40), "%s", text variable: DALI_Commissioning.fbPart102Scenes.nScene
        OnMouseClick: write the text variable via Default, min 0, max 15, title "Choose scene"
    Group (10,5 170x40)
        Textfield (0,0 110x40), "DALI Line:"
        Button (90,0 80x40), "%d", text variable: GVL_Internal.nDALILine
            OnMouseClick: write the text variable via Default, min 1, max 10, title "Choose line"
END_VISUALIZATION

// ---- POUs/DALI/DALI_Setup/VISUs/Visu_DALICommissioning/Visu_Part103Parameters.TcVIS
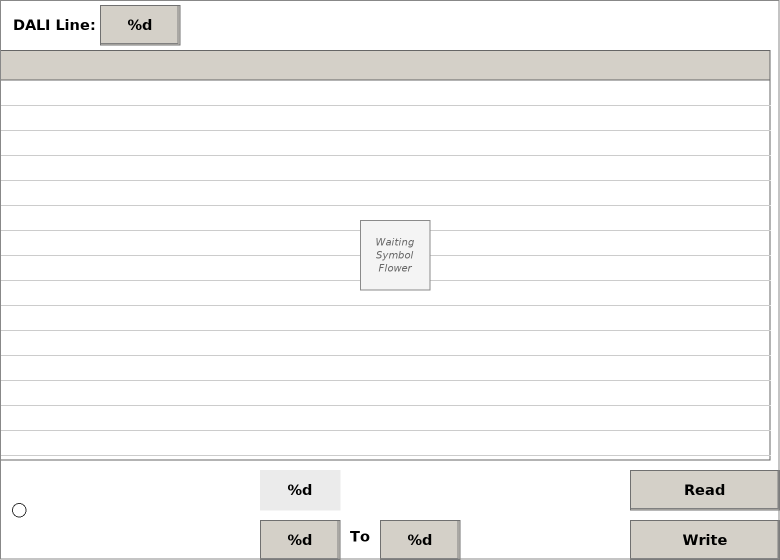
VISUALIZATION Visu_Part103Parameters  // 780x560
    Table (0,50 770x410), data array: DALI_Commissioning.fbPart103Parameters.aParameters
        p1137915858: DALI_Commissioning.fbPart103Parameters.nSelectedAddress
        p3854506369: DALI_Commissioning.fbPart103Parameters.aParameters[INDEX].nOperatingMode
        p1892666644: DALI_Commissioning.fbPart103Parameters.aParameters[INDEX].sInstanceType0
        p338671338: DALI_Commissioning.fbPart103Parameters.aParameters[INDEX].sInstanceType1
        p2170511999: DALI_Commissioning.fbPart103Parameters.aParameters[INDEX].sInstanceType2
        p3723444502: DALI_Commissioning.fbPart103Parameters.aParameters[INDEX].sInstanceType3
        p1218418051: DALI_Commissioning.fbPart103Parameters.aParameters[INDEX].sInstanceType4
        p511219082: IT0 (Generic Input)
        p1755163831: IT1 (PushButton)
        p4092479075: IT2 (Absolute Input)
        p2237128397: IT3 (Occupancy)
        p505689113: IT4 (Light Sensor)
        Columns.Column.[0].Template: OnMouseClick: write the text variable via Default, min 0, max 255, title "Insert Operating Mode 0, 128-255"
    RadioButton (10,460 230x100), variable: DALI_Commissioning.fbPart103Parameters.nAddressRange
        Areas[0]: Text=Single Short Address
        Areas[1]: Text=Short Address Range
    Textfield (260,470 80x40), "%d", text variable: DALI_Commissioning.fbPart103Parameters.nSelectedAddress
    Button (260,520 80x40), "%d", text variable: DALI_Commissioning.fbPart103Parameters.nStartAddress
        OnMouseClick: write the text variable via Default, min 0, max 63, title "Insert Short Address"
    Button (380,520 80x40), "%d", text variable: DALI_Commissioning.fbPart103Parameters.nEndAddress
        OnMouseClick: write the text variable via Default, min 0, max 63, title "Insert Short Address"
    Button (630,470 150x40), "Read"
        OnMouseClick: execute { DALI_Commissioning.fbPart103Parameters.bRead := true; }
    Button (630,520 150x40), "Write"
        OnMouseClick: execute { DALI_Commissioning.fbPart103Parameters.bWrite := true; }
    Textfield (335,521 50x31), "To"
    WaitingSymbolFlower (360,220 70x70), invisible if: DALI_Commissioning.fbPart103Parameters.bHideWaitSymbol
    Group (10,5 170x40)
        Textfield (0,0 110x40), "DALI Line:"
        Button (90,0 80x40), "%d", text variable: GVL_Internal.nDALILine
            OnMouseClick: write the text variable via Default, min 1, max 10, title "Choose line"
END_VISUALIZATION

// ---- POUs/DALI/DALI_Setup/VISUs/Visu_DALICommissioning/Visu_Part202Status.TcVIS
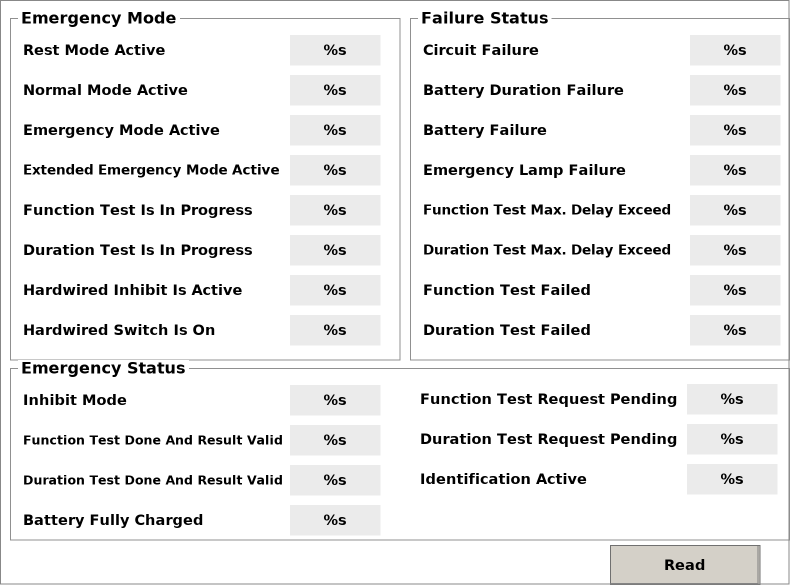
VISUALIZATION Visu_Part202Status  // 790x585
    Button (610,545 150x40), "Read"
        OnMouseClick: execute { DALI_Commissioning.fbPart202Emergency.bReadState:=TRUE; }
    GroupBox (10,10 390x350), "Emergency Mode"
        Textfield (10,145 260x30), "Extended Emergency Mode Active"
        Textfield (280,185 90x30), "%s", text variable: DALI_Commissioning.fbPart202Emergency.sFunctionTest
        Textfield (280,145 90x30), "%s", text variable: DALI_Commissioning.fbPart202Emergency.sExtendedEmergency
        Textfield (280,105 90x30), "%s", text variable: DALI_Commissioning.fbPart202Emergency.sEmergencyMode
        Textfield (280,65 90x30), "%s", text variable: DALI_Commissioning.fbPart202Emergency.sNormalMode
        Textfield (280,25 90x30), "%s", text variable: DALI_Commissioning.fbPart202Emergency.sRestMode
        Textfield (10,25 260x30), "Rest Mode Active"
        Textfield (10,65 260x30), "Normal Mode Active"
        Textfield (10,105 260x30), "Emergency Mode Active"
        Textfield (10,185 260x30), "Function Test Is In Progress"
        Textfield (10,225 260x30), "Duration Test Is In Progress"
        Textfield (10,265 260x30), "Hardwired Inhibit Is Active"
        Textfield (10,305 260x30), "Hardwired Switch Is On"
        Textfield (280,265 90x30), "%s", text variable: DALI_Commissioning.fbPart202Emergency.sHardwiredInhibit
        Textfield (280,305 90x30), "%s", text variable: DALI_Commissioning.fbPart202Emergency.sHardwiredSwitch
        Textfield (280,225 90x30), "%s", text variable: DALI_Commissioning.fbPart202Emergency.sDurationTest
    GroupBox (410,10 380x350), "Failure Status"
        Textfield (10,145 260x30), "Emergency Lamp Failure"
        Textfield (280,185 90x30), "%s", text variable: DALI_Commissioning.fbPart202Emergency.sFunctionTestExceed
        Textfield (280,145 90x30), "%s", text variable: DALI_Commissioning.fbPart202Emergency.sEmergencyLampFailure
        Textfield (280,105 90x30), "%s", text variable: DALI_Commissioning.fbPart202Emergency.sBatteryFailure
        Textfield (280,65 90x30), "%s", text variable: DALI_Commissioning.fbPart202Emergency.sBatteryDurationFailure
        Textfield (280,25 90x30), "%s", text variable: DALI_Commissioning.fbPart202Emergency.sCircuitFailure
        Textfield (10,25 260x30), "Circuit Failure"
        Textfield (10,65 260x30), "Battery Duration Failure"
        Textfield (10,105 260x30), "Battery Failure"
        Textfield (10,185 260x30), "Function Test Max. Delay Exceed"
        Textfield (10,225 260x30), "Duration Test Max. Delay Exceed"
        Textfield (10,265 260x30), "Function Test Failed"
        Textfield (10,305 260x30), "Duration Test Failed"
        Textfield (280,265 90x30), "%s", text variable: DALI_Commissioning.fbPart202Emergency.sFunctionTestFailed
        Textfield (280,305 90x30), "%s", text variable: DALI_Commissioning.fbPart202Emergency.sDurationTestFailed
        Textfield (280,225 90x30), "%s", text variable: DALI_Commissioning.fbPart202Emergency.sDurationTestExceed
    GroupBox (10,360 780x180), "Emergency Status"
        Textfield (10,145 260x30), "Battery Fully Charged"
        Textfield (677,24 90x30), "%s", text variable: DALI_Commissioning.fbPart202Emergency.sFunctionTestRequestPending
        Textfield (10,25 260x30), "Inhibit Mode"
        Textfield (10,65 260x30), "Function Test Done And Result Valid"
        Textfield (407,24 260x30), "Function Test Request Pending"
        Textfield (407,64 260x30), "Duration Test Request Pending"
        Textfield (407,104 260x30), "Identification Active"
        Textfield (677,104 90x30), "%s", text variable: DALI_Commissioning.fbPart202Emergency.sIdentificationActive
        Textfield (677,64 90x30), "%s", text variable: DALI_Commissioning.fbPart202Emergency.sDurationTestRequestPending
        Textfield (280,25 90x30), "%s", text variable: DALI_Commissioning.fbPart202Emergency.sInhibitMode
        Textfield (280,65 90x30), "%s", text variable: DALI_Commissioning.fbPart202Emergency.sFunctionTestDoneValid
        Textfield (280,145 90x30), "%s", text variable: DALI_Commissioning.fbPart202Emergency.sBatteryFullCharged
        Textfield (10,105 260x30), "Duration Test Done And Result Valid"
        Textfield (280,105 90x30), "%s", text variable: DALI_Commissioning.fbPart202Emergency.sDurationTestDoneValid
END_VISUALIZATION

// ---- POUs/DALI/DALI_Setup/VISUs/Visu_DALICommissioning/Visu_Part302AbsoluteInputDevice.TcVIS
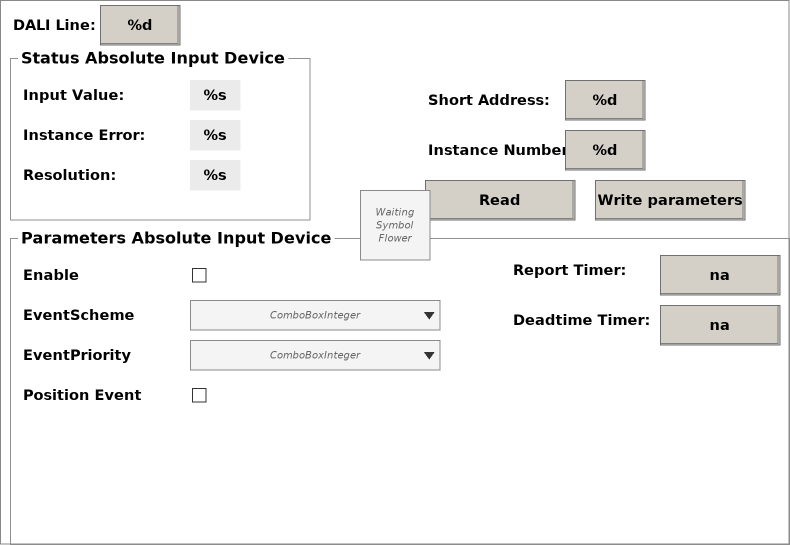
VISUALIZATION Visu_Part302AbsoluteInputDevice  // 790x545
    GroupBox (10,50 300x170), "Status Absolute Input Device"
        Textfield (10,30 160x30), "Input Value:"
        Textfield (10,70 160x30), "Instance Error:"
        Textfield (10,110 160x30), "Resolution:"
        Textfield (180,30 50x30), "%s", text variable: DALI_Commissioning.fbPart302AbsoluteInputDevice.nInputValue
        Textfield (180,70 50x30), "%s", text variable: DALI_Commissioning.fbPart302AbsoluteInputDevice.nInstanceError
        Textfield (180,110 50x30), "%s", text variable: DALI_Commissioning.fbPart302AbsoluteInputDevice.nResolution
    Button (425,180 150x40), "Read"
        OnMouseClick: execute { DALI_Commissioning.fbPart302AbsoluteInputDevice.bRead := TRUE; }
    GroupBox (10,230 780x315), "Parameters Absolute Input Device"
        Textfield (500,75 145x30), "Deadtime Timer:"
        Textfield (500,25 145x30), "Report Timer:"
        Textfield (10,30 150x30), "Enable"
        Button (650,25 120x40), "%d s", text variable: DALI_Commissioning.fbPart302AbsoluteInputDevice.nReport
            OnMouseClick: write DALI_Commissioning.fbPart302AbsoluteInputDevice.nReport via Default, min 0, max 255, title "Insert value for report timer"
        Button (650,75 120x40), "%d ms", text variable: DALI_Commissioning.fbPart302AbsoluteInputDevice.nDeadtime
            OnMouseClick: write DALI_Commissioning.fbPart302AbsoluteInputDevice.nDeadtime via Default, min 0, max 12750, title "Insert value for deadtime timer"
        Checkbox (180,30 30x30), variable: DALI_Commissioning.fbPart302AbsoluteInputDevice.bEnable
        Textfield (10,70 150x30), "EventScheme"
        ComboBoxInteger (180,70 250x30), variable: DALI_Commissioning.fbPart302AbsoluteInputDevice.eEventScheme, text list: 'EventScheme'
        Button (650,25 120x40), "na", invisible if: Not DALI_Commissioning.fbPart302AbsoluteInputDevice.bNoReportTimer, input disabled if: Not DALI_Commissioning.fbPart302AbsoluteInputDevice.bNoReportTimer
        Button (650,75 120x40), "na", invisible if: Not DALI_Commissioning.fbPart302AbsoluteInputDevice.bNoDeadtimeTimer, input disabled if: Not DALI_Commissioning.fbPart302AbsoluteInputDevice.bNoDeadtimeTimer
        Textfield (10,110 150x30), "EventPriority"
        Textfield (10,150 150x30), "Position Event"
        ComboBoxInteger (180,110 250x30), variable: DALI_Commissioning.fbPart302AbsoluteInputDevice.eEventPriority, text list: 'EventPriority'
        Checkbox (180,150 30x30), variable: DALI_Commissioning.fbPart302AbsoluteInputDevice.bPositionEventEnabled
    WaitingSymbolFlower (360,190 70x70), invisible if: DALI_Commissioning.fbPart302AbsoluteInputDevice.bHideWaitSymbol
    Button (595,180 150x40), "Write parameters"
        OnMouseClick: execute { DALI_Commissioning.fbPart302AbsoluteInputDevice.bWrite := TRUE; }
    Group (10,5 170x40)
        Textfield (0,0 110x40), "DALI Line:"
        Button (90,0 80x40), "%d", text variable: GVL_Internal.nDALILine
            OnMouseClick: write the text variable via Default, min 1, max 10, title "Choose line"
    Textfield (425,80 130x40), "Short Address:"
    Button (565,80 80x40), "%d", text variable: DALI_Commissioning.fbPart302AbsoluteInputDevice.nAddress
        OnMouseClick: write DALI_Commissioning.fbPart302AbsoluteInputDevice.nAddress via Default, min 0, max 63, title "Insert Short Address"
    Textfield (425,130 150x40), "Instance Number:"
    Button (565,130 80x40), "%d", text variable: DALI_Commissioning.fbPart302AbsoluteInputDevice.nInstanceAddress
        OnMouseClick: write DALI_Commissioning.fbPart302AbsoluteInputDevice.nInstanceAddress via Default, min 0, max 31, title "Insert instance number"
END_VISUALIZATION
